TYPE ST_CSL_Colors :
STRUCT
	aRed 	: 	ARRAY[0 .. 1] TO REAL;
	aWhite 	: 	ARRAY[0 .. 1] TO REAL;
	aBlue 	: 	ARRAY[0 .. 1] TO REAL;
END_STRUCT
END_TYPE

(* stored: Version 1.1.0.1, ProductVersion 3.1.4024.12
   DUT ST_CSL_Colors: Id {5d213f91-e3d6-4af4-b4c6-7b625ccf3af6} *)
